TYPE ST_System_BSp_Verb_Parameter :
STRUCT
	AutoQuittierung			: BOOL := 0;
	Kennlinie_Tctr			: DINT := 5000;
    Temp_Durchmischung 		: REAL ; (*Wenn die Temperatur mehr als dieser Wert ist, dann darf die Pumpe zur Durchmischung angeschaltet werden*)


END_STRUCT
END_TYPE

(* stored: Version 1.1.0.1, ProductVersion 3.1.4024.9
   DUT ST_System_BSp_Verb_Parameter: Id {12e5514c-c5da-4e83-a8d7-f248cd617088} *)
